# EPICS autosave request: iocBoot/gmca_23b_ioc1/dbSave/GO_Om_.req
%
% BURT Request File
%
% $(P)GO:Om:  Goniometer Omega
%

file assy.req ASSY=$(P)GO:Om
file mtr1.req MTR1=$(P)GO:mom
file drv1.req DRV1=$(P)GO:OM
